(* Schneider Machine Expert - Basic project Traffic, file version 1.6.0.0 *)
(* ProjectInformations: Name=New project *)

HARDWARE
  Cpu 0: TM221CE16R
  EthernetConfiguration: NetworkName=M221, IpAllocationMode=FixedAddress, IpAddress=0.0.0.0, SubnetMask=0.0.0.0
  SerialLineConfiguration: Baud=Baud19200, Parity=ParityEven, DataBits=DataBits8, StopBits=StopBits1, PhysicalMedium=PhysicalMediumRs485, TransmissionMode=TransmissionModeModbusRtu, SlaveId=1, Addressing=SlaveAddressing
  MastTask: UsePeriodScanMode=false, PeriodScan=100
  FastTask: Period=255
  CpuBehavior: StartingMode=StartAsPreviousState, AutoSaveRamOnEeprom=true, WatchdogPeriod=250

SYMBOLS  (address, symbol, comment, settings)
  %TM0        [Type=TP, Preset=3, Base=OneSecond]
  %TM1        [Type=TOF, Preset=5, Base=OneSecond]
  %TM2        [Preset=2, Base=OneSecond]
  %TM3        [Preset=5, Base=OneHundredMilliSeconds]

POU New POU
  (* SectionNumber=1 *)

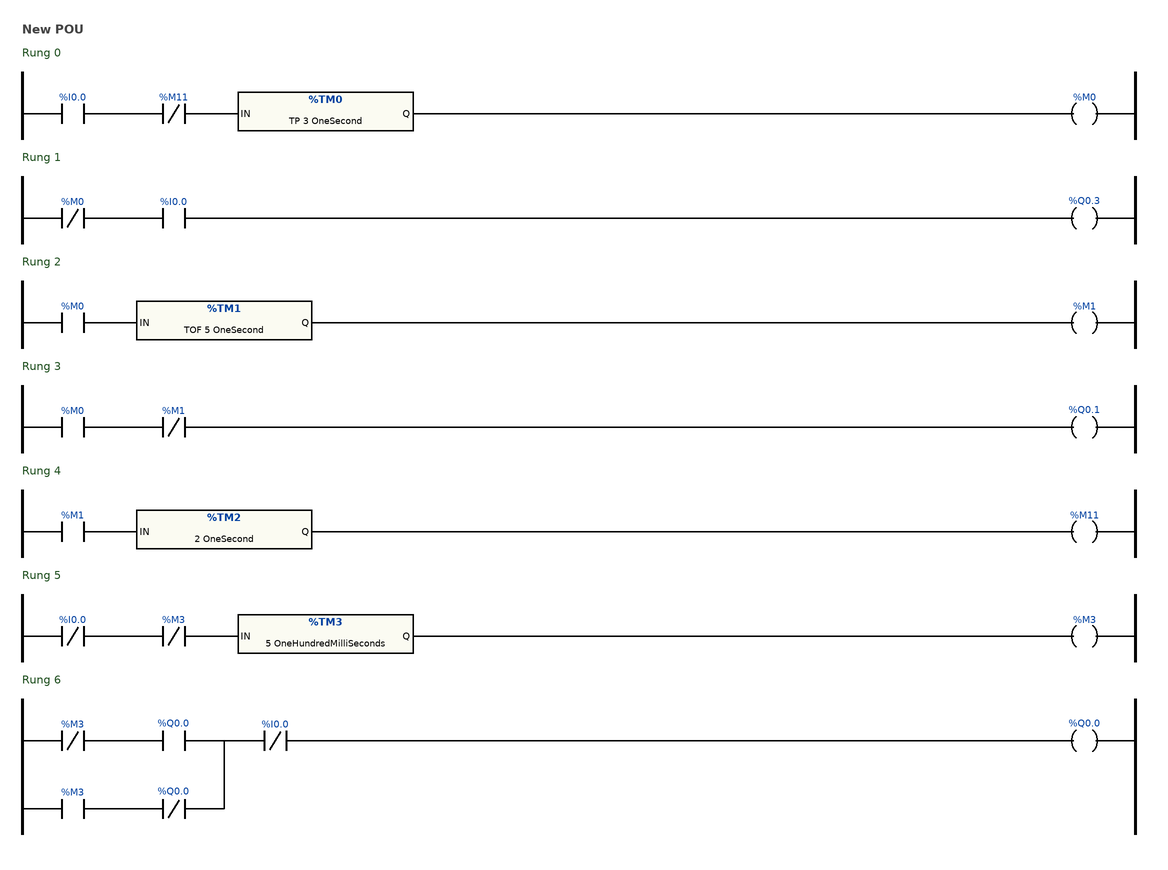

// Rung 0
  BLK %TM0
  LD %I0.0
  ANDN %M11
  IN
  OUT_BLK
  LD Q
  ST %M0
  END_BLK
  // as ST:
  //   %TM0(IN := %I0.0 AND NOT %M11);
  //   %M0 := %TM0.Q;

// Rung 1
  LDN %M0
  AND %I0.0
  ST %Q0.3
  // as ST:
  //   %Q0.3 := NOT %M0 AND %I0.0;

// Rung 2
  BLK %TM1
  LD %M0
  IN
  OUT_BLK
  LD Q
  ST %M1
  END_BLK
  // as ST:
  //   %TM1(IN := %M0);
  //   %M1 := %TM1.Q;

// Rung 3
  LD %M0
  ANDN %M1
  ST %Q0.1
  // as ST:
  //   %Q0.1 := %M0 AND NOT %M1;

// Rung 4
  BLK %TM2
  LD %M1
  IN
  OUT_BLK
  LD Q
  ST %M11
  END_BLK
  // as ST:
  //   %TM2(IN := %M1);
  //   %M11 := %TM2.Q;

// Rung 5
  BLK %TM3
  LDN %I0.0
  ANDN %M3
  IN
  OUT_BLK
  LD Q
  ST %M3
  END_BLK
  // as ST:
  //   %TM3(IN := NOT %I0.0 AND NOT %M3);
  //   %M3 := %TM3.Q;

// Rung 6
  LDN %M3
  AND %Q0.0
  OR( %M3
  ANDN %Q0.0
  )
  ANDN %I0.0
  ST %Q0.0
  // as ST:
  //   %Q0.0 := (NOT %M3 AND %Q0.0 OR %M3 AND NOT %Q0.0) AND NOT %I0.0;
